Staubli VAL3: exit.pgx

program exit()
begin
  bExit = true
end
